FUNCTION_BLOCK SpeedTrigger EXTENDS Objective IMPLEMENTS iObjective
VAR_INPUT

	ThresholdVelocity	: LREAL;

END_VAR
VAR_OUTPUT
	MoverInVelocity		: BOOL;
END_VAR
VAR
	someMoverInVelo: BOOL;
	whichMover: INT;
	i: INT;
END_VAR



MonitorSuccesses();

METHOD Cyclic : BOOL
VAR_INPUT
END_VAR
END_METHOD

ACTION MonitorSuccesses:


someMoverInVelo		:= FALSE;
whichMover			:= 0;

FOR i := 0 TO GVL.NUM_MOVERS-1 DO
	
	IF TrackedMovers[i] <> 0 THEN
		
		IF (ABS(TrackedMovers[i]^.AxisReference.NcToPlc.ActVelo) >= ThresholdVelocity) THEN
			someMoverInVelo		:= TRUE;
			whichMover			:= i; 
		END_IF
	END_IF
	
END_FOR

IF someMoverInVelo THEN
	MoverInVelocity			:= TRUE;
//	CurrentMover			REF= TrackedMovers[whichMover]^;
ELSE
	MoverInVelocity			:= FALSE;
//	CurrentMover			REF= 0;		
END_IF
END_ACTION

END_FUNCTION_BLOCK

(* stored: Version 1.1.0.1, ProductVersion 3.1.4024.9
   POU SpeedTrigger: Id {ceb84e98-9bb3-44af-9526-f95d6c0344e5}, SpecialFunc None
   Folder Methods: Id {23916c1a-8736-47b3-84aa-78b43be3b9c9}
   Folder Properties: Id {1b5810cd-1bcb-4f24-a665-f771a8e481c0}
   Method Cyclic: Id {c99ce270-5c9c-450e-a563-d1b16d69ceec}
   Action MonitorSuccesses: Id {69f23fdc-e801-422e-9739-ad286b1f7aed} *)
